// TIA Portal V17 export
// export: Created 2025-03-07T09:19:58.5465715Z, ExportSetting WithDefaults, DisplayName Totally Integrated Automation Portal, DisplayVersion V17 Update 8, DisplayName TIA Portal Openness, DisplayVersion V17 Update 8, DisplayName TIA Portal Version Control Interface, DisplayVersion V17, DisplayName SINAMICS Startdrive Advanced, DisplayVersion V17 SP2, DisplayName SINAMICS Startdrive G110M, G120, G120C, G120D, G120P, G115D, DisplayVersion V17 SP2, DisplayName SINAMICS Startdrive G130, G150, S120, S150, SINAMICS MV, S210, DisplayVersion V17 SP2, DisplayName STEP 7 Professional, DisplayVersion V17 Update 8, DisplayName SINUMERIK ONE STEP 7 Toolbox, DisplayVersion V17 Update 12, DisplayName SINUMERIK 840D sl STEP 7 Toolbox, DisplayVersion V17 Update 12, DisplayName STEP 7 Safety, DisplayVersion V17 Update 6, DisplayName WinCC Advanced, DisplayVersion V17 Update 8
TYPE "POWDER FEEDER INTERLOCK OUTPUT"
// stored: IsFailsafeCompliant false
   STRUCT
      o_uiOperationMode : Word;   // Operation Mode 0 = Standalone, 1 = On Off Remote 2 = UDP, 3 = Profibus / operation mode 2 = UDP, 3 = Profibus, 4 = ProfiNet
      Spare_Word_0 : Word;   // Spare
      o_uiProductionMode : Word;   // Production Mode 0 = Off, 1 = Production / production mode 0 = OFF, 1 = Production
      Spare_Word_1 : Word;   // Spare
      o_uiSystemMode : Word;   // 0 = Plasma 1 = HVOF
      Spare_Word_2 : Word;   // Spare
      o_fAirFlowIsRunning : Bool;   // 0 = No Airflow, 1 = Airflow Present / 0 = no airflow, 1 = Airflow present
      o_fCarrierGasSelect : Bool;   // 0 = Carrier Gas Argon, 1 = Carrier Gas Nitrogen / 0 = carriergas Argon, 1 = carriergas Nitrogen
      o_fUnitSelect : Bool;   // 0 = Metric, 1 = SI / 0 = metric, 1 = SI
      Spare_0 : Bool;   // Spare
      Spare_1 : Bool;   // Spare
      Spare_2 : Bool;   // Spare
      Spare_3 : Bool;   // Spare
      Spare_4 : Bool;   // Spare
      o_fVolumetricMode_Line1 : Bool;   // 1 = Volumetric Mode On / 1 = volumetric mode on
      o_fVolumetricMode_Line2 : Bool;   // 1 = Volumetric Mode On / 1 = volumetric mode on
      o_fGravimetricMode_Line1 : Bool;   // 1 = Gravimetric Mode On n/a for Twin 150 / 1 = gravimetric mode on n/a for Twin 150
      o_fGravimetricMode_Line2 : Bool;   // 1 = Gravimetric Mode On n/a for Twin 150 / 1 = gravimetric mode on n/a for Twin 150
      o_fTareCmd_Line1 : Bool;   // N/a For Twin 150 / n/a for Twin 150
      o_fTareCmd_Line2 : Bool;   // N/a For Twin 150 / n/a for Twin 150
      Spare_5 : Bool;   // Spare
      Spare_6 : Bool;   // Spare
      o_fCalibCmd_Line1 : Bool;   // N/a For Twin 150 / n/a for Twin 150
      o_fCalibCmd_Line2 : Bool;   // N/a For Twin 150 / n/a for Twin 150
      Spare_7 : Bool;   // Spare
      Spare_8 : Bool;   // Spare
      o_fShutdownToPF_Line1 : Bool;   // 0 = Controller Doesn't Request Shutdown / 0 = controller doesn't request shutdown, 1 = controller requests shutdown
      o_fShutdownToPF_Line2 : Bool;   // 1 = Controller Requests Shutdown / 0 = controller doesn't request shutdown, 1 = controller requests shutdown
      o_fCommunicationOk_Line1 : Bool;   // Communication Is Running / Communication is running
      o_fCommunicationOk_Line2 : Bool;   // Communication Is Running / Communication is running
      o_fFeedingAllOnCmd_Line1 : Bool;   // 1 = Start Stirrer & Disk (Pos. Edge Trigger) / 1 = start stirrer & disk (pos. Edge trigger)
      o_fFeedingAllOnCmd_Line2 : Bool;   // 1 = Start Stirrer & Disk (Pos. Edge Trigger) / 1 = start stirrer & disk (pos. Edge trigger)
      o_fCarriergasOnCmd_Line1 : Bool;   // 1 = Start Carrier Gas / 1 = start carriergas (pos. Edge trigger)
      o_fCarriergasOnCmd_Line2 : Bool;   // 1 = Start Carrier Gas / 1 = start carriergas (pos. Edge trigger)
      o_fFeedingAllOffCmd_Line1 : Bool;   // 1 = Stop Stirrer & Disk / 1 = stop stirrer & disk
      o_fFeedingAllOffCmd_Line2 : Bool;   // 1 = Stop Stirrer & Disk / 1 = stop stirrer & disk
      o_fCarriergasOffCmd_Line1 : Bool;   // 1 = Stop Carrier Gas / 1 = stop carriergas
      o_fCarriergasOffCmd_Line2 : Bool;   // 1 = Stop Carrier Gas / 1 = stop carriergas
      o_fHeatingOnCmd_Line1 : Bool;   // 1 = Start Heating (Pos. Edge Trigger) / 1 = start heating (pos. Edge trigger)
      o_fHeatingOnCmd_Line2 : Bool;   // 1 = Start Heating (Pos. Edge Trigger) / 1 = start heating (pos. Edge trigger)
      o_fHeatingOffCmd_Line1 : Bool;   // 1 = Stop Heating / 1 = stop heating
      o_fHeatingOffCmd_Line2 : Bool;   // 1 = Stop Heating / 1 = stop heating
      Spare_9 : Bool;   // Spare
      Spare_10 : Bool;   // Spare
      Spare_11 : Bool;   // Spare
      Spare_12 : Bool;   // Spare
      Spare_Byte_0 : Byte;   // Spare
      Spare_Byte_1 : Byte;   // Spare
      Spare_Byte_2 : Byte;   // Spare
      "PF Setpoints, Warnings and Alarms" : Struct
         o_rCarriergasNominal_Line1 : Real;   // Carrier Gas Setpoint [NLPM] (0..16 NLPM) / carriergas setpoint [NLPM] (0..16 NLPM)
         o_rCarriergasNominal_Line2 : Real;   // Carrier Gas Setpoint [NLPM] (0..16 NLPM) / carriergas setpoint [NLPM] (0..16 NLPM)
         o_rDiskSpeedNominal_Line1 : Real;   // Disk Speed Setpoint [%] (0..100 %) / Disk speed setpoint [%] (0..100 %)
         o_rDiskSpeedNominal_Line2 : Real;   // Disk Speed Setpoint [%] (0..100 %) / Disk speed setpoint [%] (0..100 %)
         o_rStirrerSpeedNominal_Line1 : Real;   // Stirrer Speed Setpoint [%] (30 - 100%) / Stirrer speed setpoint [%] (30 - 100%)
         o_rStirrerSpeedNominal_Line2 : Real;   // Stirrer Speed Setpoint [%] (30 - 100%) / Stirrer speed setpoint [%] (30 - 100%)
         o_rFeedrateNominal_Line1 : Real;   // N/a For Twin 150 / n/a for Twin 150
         o_rFeedrateNominal_Line2 : Real;   // N/a For Twin 150 / n/a for Twin 150
         o_rHopperTempNominal_Line1 : Real;   // Hopper Temperature Setpoint [°C] (n/a for Twin 150 R1.0) / Hopper temperature setpoint [°C]
         o_rHopperTempNominal_Line2 : Real;   // Hopper Temperature Setpoint [°C] (n/a for Twin 150 R1.0) / Hopper temperature setpoint [°C]
         o_rLoadcellCalibrationNominal_Line1 : Real;   // N/a For Twin 150 / n/a for Twin 150
         o_rLoadcellCalibrationNominal_Line2 : Real;   // N/a For Twin 150 / n/a for Twin 150
         o_rPowderFactorNominal_Line1 : Real;   // N/a For Twin 150 / n/a for Twin 150
         o_rPowderFactorNominal_Line2 : Real;   // N/a For Twin 150 / n/a for Twin 150
         o_rLLlimitCarriergas_Line1 : Real;   // Carrier Gas Flow LL Limit [NLPM] (Absolute Value) / carriergas flow LL limit [NLPM] (absolute value)
         o_rLLlimitCarriergas_Line2 : Real;   // Carrier Gas Flow LL Limit [NLPM] (Absolute Value) / carriergas flow LL limit [NLPM] (absolute value)
         o_rLLlimitDiskSpeedNominal_Line1 : Real;   // Disk Speed LL Limit [%] (Absolute Value) / Disk speed LL limit [%] (absolute value)
         o_rLLlimitDiskSpeedNominal_Line2 : Real;   // Disk Speed LL Limit [%] (Absolute Value) / Disk speed LL limit [%] (absolute value)
         o_rLLlimitStirrerSpeedNominal_Line1 : Real;   // Stirrer Speed LL Limit [%] (Absolute Value) / Stirrer speed LL limit [%] (absolute value)
         o_rLLlimitStirrerSpeedNominal_Line2 : Real;   // Stirrer Speed LL Limit [%] (Absolute Value) / Stirrer speed LL limit [%] (absolute value)
         o_rLLlimitFeedRateNominal_Line1 : Real;   // N/a For Twin 150 / n/a for Twin 150
         o_rLLlimitFeedRateNominal_Line2 : Real;   // N/a For Twin 150 / n/a for Twin 150
         o_rLlimitCarriergas_Line1 : Real;   // Carrier Gas L Limit [NLPM] (Absolute Value) / carriergas L limit [NLPM] (absolute value)
         o_rLlimitCarriergas_Line2 : Real;   // Carrier Gas L Limit [NLPM] (Absolute Value) / carriergas L limit [NLPM] (absolute value)
         o_rLlimitDiskSpeedNominal_Line1 : Real;   // Disk Speed L Limit [%] (Absolute Value) / Disk speed L limit [%] (absolute value)
         o_rLlimitDiskSpeedNominal_Line2 : Real;   // Disk Speed L Limit [%] (Absolute Value) / Disk speed L limit [%] (absolute value)
         o_rLlimitStirrerSpeedNominal_Line1 : Real;   // Stirrer Speed L Limit [%] (Absolute Value) / Stirrer speed L limit [%] (absolute value)
         o_rLlimitStirrerSpeedNominal_Line2 : Real;   // Stirrer Speed L Limit [%] (Absolute Value) / Stirrer speed L limit [%] (absolute value)
         o_rLlimitFeedRateNominal_Line1 : Real;   // N/a For Twin 150 / n/a for Twin 150
         o_rLlimitFeedRateNominal_Line2 : Real;   // N/a For Twin 150 / n/a for Twin 150
         o_rHlimitCarriergas_Line1 : Real;   // Carrier Gas H Limit [NLPM] (Absolute Value) / Carriergas H limit [NLPM] (absolute value)
         o_rHlimitCarriergas_Line2 : Real;   // Carrier Gas H Limit [NLPM] (Absolute Value) / Carriergas H limit [NLPM] (absolute value)
         o_rHlimitDiskSpeedNominal_Line1 : Real;   // Disk Speed H Limit [%] (Absolute Value) / Disk speed H limit [%] (absolute value)
         o_rHlimitDiskSpeedNominal_Line2 : Real;   // Disk Speed H Limit [%] (Absolute Value) / Disk speed H limit [%] (absolute value)
         o_rHlimitStirrerSpeedNominal_Line1 : Real;   // Stirrer Speed H Limit [%] (Absolute Value) / Stirrer speed H limit [%] (absolute value)
         o_rHlimitStirrerSpeedNominal_Line2 : Real;   // Stirrer Speed H Limit [%] (Absolute Value) / Stirrer speed H limit [%] (absolute value)
         o_rHlimitFeedRateNominal_Line1 : Real;   // N/a For Twin 150 / n/a for Twin 150
         o_rHlimitFeedRateNominal_Line2 : Real;   // N/a For Twin 150 / n/a for Twin 150
         o_rHHlimitCarriergas_Line1 : Real;   // Carrier Gas HH Limit [NLPM] (Absolute Value) / Carriergas HH limit [NLPM] (absolute value)
         o_rHHlimitCarriergas_Line2 : Real;   // Carrier Gas HH Limit [NLPM] (Absolute Value) / Carriergas HH limit [NLPM] (absolute value)
         o_rHHlimitDiskSpeedNominal_Line1 : Real;   // Disk Speed HH Limit [%] (Absolute Value) / Disk speed HH limit [%] (absolute value)
         o_rHHlimitDiskSpeedNominal_Line2 : Real;   // Disk Speed HH Limit [%] (Absolute Value) / Disk speed HH limit [%] (absolute value)
         o_rHHlimitStirrerSpeedNominal_Line1 : Real;   // Stirrer Speed HH Limit [%] (Absolute Value) / Stirrer speed HH limit [%] (absolute value)
         o_rHHlimitStirrerSpeedNominal_Line2 : Real;   // Stirrer Speed HH Limit [%] (Absolute Value) / Stirrer speed HH limit [%] (absolute value)
         o_rHHlimitFeedRateNominal_Line1 : Real;   // N/a For Twin 150 / n/a for Twin 150
         o_rHHlimitFeedRateNominal_Line2 : Real;   // N/a For Twin 150 / n/a for Twin 150
         o_rHHlimitHopperTempNominal_Line1 : Real;   // Hopper Temperature HH Limit (ºC), (Absolute Value, N/a For Twin 150 R1.0) / Hopper temperature HH limit [°C] (absolute value, n/a for Twin 150)
         o_rHHlimitHopperTempNominal_Line2 : Real;   // Hopper Temperature HH Limit (ºC), (Absolute Value, N/a For Twin 150 R1.0) / Hopper temperature HH limit [°C] (absolute value, n/a for Twin 150)
      END_STRUCT;
   END_STRUCT;
END_TYPE
